{attribute 'linkalways'}
{attribute 'no_explicit_call' := 'do not call this POU directly'}
FUNCTION_BLOCK RegisterInstanceToTaskCallback IMPLEMENTS I_Callback
VAR
	task : I_Task;
END_VAR

METHOD FB_init : BOOL
VAR_INPUT
	bInitRetains : BOOL; // if TRUE, the retain variables are initialized (warm start / cold start)
	bInCopyCode : BOOL;  // if TRUE, the instance afterwards gets moved into the copy code (online change)
	Task : I_Task;
END_VAR
this^.task := Task;
END_METHOD

METHOD PUBLIC Update
VAR_INPUT
	event : I_Event;
END_VAR
VAR
	instanceAdded : I_InstanceAddedEvent;
END_VAR
IF NOT __QUERYINTERFACE(event, instanceAdded) THEN
	RETURN;
END_IF

IF task.SharesNamespaceWith(instanceAdded.Instance) THEN
	task.RegisterInstance(instanceAdded.Instance);
	RETURN;
END_IF

IF task.IsExecutingThis() THEN
	task.RegisterInstance(instanceAdded.Instance);
	RETURN;
END_IF
END_METHOD

END_FUNCTION_BLOCK

(* stored: Version 1.1.0.1, ProductVersion 3.1.4024.11
   POU RegisterInstanceToTaskCallback: Id {c97dc573-b0a5-43aa-b12e-6ec9bfcfdd9a}, SpecialFunc None
   Folder Constructor: Id {0cc29fe1-7917-4191-9f79-b0884551051a}
   Method FB_init: Id {29bf26f7-cb05-481b-ac98-5a0ed955ecf0}
   Method Update: Id {cba2c69d-0931-4389-8631-872ff9a68c9a} *)
